(* PLC project Testimplementierung26042021.project, CODESYS CODESYS V3.5 SP16 Patch 1 *)
(* stored: creationDateTime 2021-05-02T21:54:17.2089195, modificationDateTime 2021-05-02T21:40:12.2319923 *)

PROGRAM PLC_PRG
  VAR
    taschenrechner1 : Taschenrechner;
  END_VAR

                    taschenrechner1();
                  
END_PROGRAM

FUNCTION_BLOCK Taschenrechner EXTENDS TJ.Skill
  VAR_INPUT
    zahlA : TJ.SkillParameter := (default := 5, value := 20, name := 'Zahl_A', paramType := 'INTEGER', required := TRUE);
    zahlB : TJ.SkillParameter := (default := 5, value := 20, name := 'Zahl_A', paramType := 'INTEGER', required := TRUE);
  END_VAR
  VAR_OUTPUT
    ergebnis : TJ.SkillParameter := (default := 0, value := 0, name := 'Ergebnis', paramType := 'INTEGER', required := FALSE);
  END_VAR

                    SUPER^();
                  

METHOD execute : BOOL
                          THIS^.ergebnis.value:= THIS^.zahlA.value+THIS^.zahlB.value;
completeActualState();
                        
END_METHOD
END_FUNCTION_BLOCK

CONFIGURATION Device
  RESOURCE Application ON PLC
    TASK MainTask(INTERVAL := T#20ms, PRIORITY := 1);
    PROGRAM PLC_PRG WITH MainTask : PLC_PRG;
  END_RESOURCE
END_CONFIGURATION
